Staubli VAL3: memory_path.pgx

program memory_path(string x_sPath (dimensions=1), string& x_sFolders[] (dimensions=1))
  local num i
  local num l_nSize
  local string l_sEmpty
  local string l_sPath
begin
  //
  // make o recursive all the path
  //
  l_sEmpty=""
  call use:stringCopy(l_sEmpty,sPath)
  libList(x_sPath,sPath)
  l_nSize=size(sPath)-1
  if sPath!=""
    for i=0 to l_nSize
      if find(sPath[i],".")==-1
        // compose
        l_sPath=x_sPath
        if x_sPath!=""
          // deepest
          x_sPath=x_sPath+"/"+sPath[i]
        else
          x_sPath=sPath[i]
        endIf
        //
        // increase the x_sFolders
        //
        if x_sFolders!=""
          insert(x_sFolders[size(x_sFolders)])
        endIf
        x_sFolders[size(x_sFolders)-1]=x_sPath
        //
        call memory_path(x_sPath,x_sFolders)
        // refresh the global variable
        l_sEmpty=""
        call use:stringCopy(l_sEmpty,sPath)
        libList(l_sPath,sPath)
        x_sPath=l_sPath
        //
      endIf
    endFor
  endIf
end
